KUKA KRL program: e_fraes1.src, e_fraes1.dat

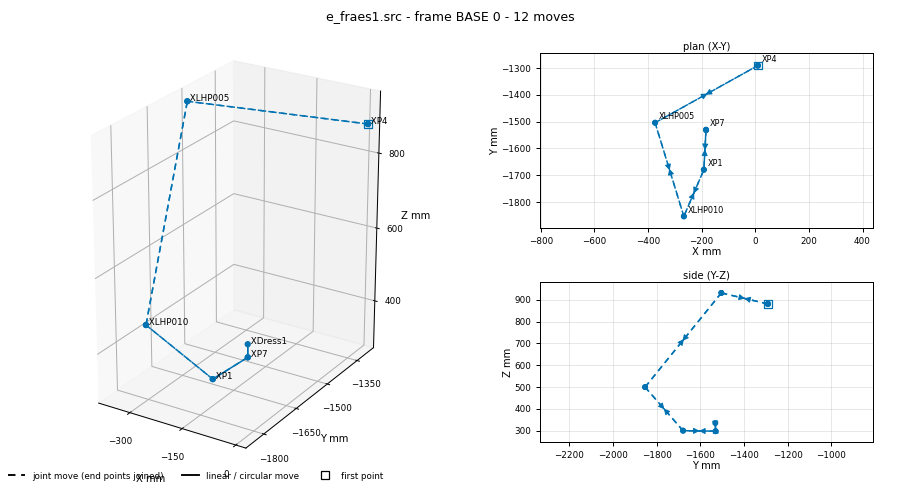
[picture p0: tool path of e_fraes1.src in frame BASE 0, 12 of 12 moves have a stored position in this frame; points joined in program order, loops and branches not executed]
--- e_fraes1.src ---
&ACCESS RVP3
&REL 71
&COMMENT Fresa C1
&PARAM DISKPATH = KRC:\R1\Program
&PARAM TEMPLATE = C:\KRC\Roboter\Template\vorgabe
&PARAM EDITMASK = *
DEF e_fraes1( )
;FOLD INI
   ;FOLD BASISTECH INI
      GLOBAL INTERRUPT DECL 3 WHEN $STOPMESS==TRUE DO IR_STOPM ( )
      INTERRUPT ON 3
      BAS (#INITMOV,0 )
   ;ENDFOLD (BASISTECH INI)
   ;FOLD SPOTTECH INI
      USERSPOT(#INIT)
   ;ENDFOLD (SPOTTECH INI)
   ;FOLD GRIPPERTECH INI
      USER_GRP(0,DUMMY,DUMMY,GDEFAULT)
   ;ENDFOLD (GRIPPERTECH INI)
   ;FOLD USER INI
      ;Make your modifications here

   ;ENDFOLD (USER INI)
;ENDFOLD (INI)

; Estacao P13.060 - Robo R2
; Programa: Fresa C1
; Caracterização dos meios de produção:
; 02/09/2014 09:15 Changes by KUKA Roboter do Brasil

chk_w1_wechs_ok () ;check c1

;FOLD Kollision.Ueberwachung_4_Ein ;%{PE}%MKUKATPUSER
COLLSTOP( 4, 1 ) ;INTERRUPTUEBERWACHT
;ENDFOLD

;FOLD PTP P4 Vel=80 % PDAT6 Tool[1]:GUN C1 Base[0];%{PE}%R 8.2.20,%MKUKATPBASIS,%CMOVE,%VPTP,%P 1:PTP, 2:P4, 3:, 5:80, 7:PDAT6
$BWDSTART=FALSE
PDAT_ACT=PPDAT6
FDAT_ACT=FP4
BAS(#PTP_PARAMS,80)
PTP XP4
;ENDFOLD
;FOLD PTP LHP005 CONT Vel=60 % PDAT2 Tool[1]:GUN C1 Base[0];%{PE}%R 8.2.20,%MKUKATPBASIS,%CMOVE,%VPTP,%P 1:PTP, 2:LHP005, 3:C_DIS, 5:60, 7:PDAT2
$BWDSTART=FALSE
PDAT_ACT=PPDAT2
FDAT_ACT=FLHP005
BAS(#PTP_PARAMS,60)
PTP XLHP005 C_DIS
;ENDFOLD
;FOLD PTP LHP010 CONT Vel= 60 % PDAT3 Tool[1]:GUN C1 Base[0];%{PE}%R 4.1.16,%MKUKATPBASIS,%CMOVE,%VPTP,%P 1:PTP, 2:LHP010, 3:C_PTP, 5:60, 7:PDAT3
$BWDSTART = FALSE
PDAT_ACT=PPDAT3
BAS(#PTP_DAT)
FDAT_ACT=FLHP010
BAS(#FRAMES)
BAS(#VEL_PTP,60)
PTP XLHP010 C_PTP
;ENDFOLD
;FOLD PTP P1 CONT Vel=60 % PDAT1 Tool[1]:GUN C1 Base[0];%{PE}%R 8.2.20,%MKUKATPBASIS,%CMOVE,%VPTP,%P 1:PTP, 2:P1, 3:C_DIS, 5:60, 7:PDAT1
$BWDSTART=FALSE
PDAT_ACT=PPDAT1
FDAT_ACT=FP1
BAS(#PTP_PARAMS,60)
PTP XP1 C_DIS
;ENDFOLD
;FOLD LIN P7 Vel=0.3 m/s CPDAT1 Tool[1]:GUN C1 Base[0];%{PE}%R 8.2.20,%MKUKATPBASIS,%CMOVE,%VLIN,%P 1:LIN, 2:P7, 3:, 5:0.3, 7:CPDAT1
$BWDSTART=FALSE
LDAT_ACT=LCPDAT1
FDAT_ACT=FP7
BAS(#CP_PARAMS,0.3)
LIN XP7
;ENDFOLD

;FOLD ; PONTO DE FRESAGEM;%{PE}%R 4.1.16,%MKUKATPBASIS,%CCOMMENT,%VNORMAL,%P 2:PONTO DE FRESAGEM
;ENDFOLD
;FOLD TIP.LIN_ Dress1, Spot Gun 1 , RETR open , Tool[1], Base[0], EXT.TCP=FALSE;%{PE}%MKUKATPUSER
FDAT_ACT=FDress1
BAS(#FRAMES)
LIN  XDress1
S_ACT.GUN=1
S_ACT.RETR=#opn
S_READY=FALSE
USERSPOT (#DRESS,S_ACT )
WAIT FOR  S_READY
;ENDFOLD

;FOLD LIN LHP020 Vel=0.3 m/s CPDAT16 Tool[1]:GUN C1 Base[0];%{PE}%R 8.2.20,%MKUKATPBASIS,%CMOVE,%VLIN,%P 1:LIN, 2:LHP020, 3:, 5:0.3, 7:CPDAT16
$BWDSTART=FALSE
LDAT_ACT=LCPDAT16
FDAT_ACT=FLHP020
BAS(#CP_PARAMS,0.3)
LIN XLHP020
;ENDFOLD
;FOLD PTP LHP025 CONT Vel= 60 % PDAT7 Tool[1]:GUN C1 Base[0];%{PE}%R 4.1.16,%MKUKATPBASIS,%CMOVE,%VPTP,%P 1:PTP, 2:LHP025, 3:C_PTP, 5:60, 7:PDAT7
$BWDSTART = FALSE
PDAT_ACT=PPDAT7
BAS(#PTP_DAT)
FDAT_ACT=FLHP025
BAS(#FRAMES)
BAS(#VEL_PTP,60)
PTP XLHP025 C_PTP
;ENDFOLD
;FOLD PTP P2 CONT Vel=60 % PDAT4 Tool[1]:GUN C1 Base[0];%{PE}%R 8.2.20,%MKUKATPBASIS,%CMOVE,%VPTP,%P 1:PTP, 2:P2, 3:C_DIS, 5:60, 7:PDAT4
$BWDSTART=FALSE
PDAT_ACT=PPDAT4
FDAT_ACT=FP2
BAS(#PTP_PARAMS,60)
PTP XP2 C_DIS
;ENDFOLD
;FOLD PTP P3 CONT Vel=60 % PDAT5 Tool[1]:GUN C1 Base[0];%{PE}%R 8.2.20,%MKUKATPBASIS,%CMOVE,%VPTP,%P 1:PTP, 2:P3, 3:C_DIS, 5:60, 7:PDAT5
$BWDSTART=FALSE
PDAT_ACT=PPDAT5
FDAT_ACT=FP3
BAS(#PTP_PARAMS,60)
PTP XP3 C_DIS
;ENDFOLD
;FOLD PTP P6 CONT Vel=60 % PDAT9 Tool[1]:GUN C1 Base[0];%{PE}%R 8.2.20,%MKUKATPBASIS,%CMOVE,%VPTP,%P 1:PTP, 2:P6, 3:C_DIS, 5:60, 7:PDAT9
$BWDSTART=FALSE
PDAT_ACT=PPDAT9
FDAT_ACT=FP6
BAS(#PTP_PARAMS,60)
PTP XP6 C_DIS
;ENDFOLD
;FOLD PTP pTEST_WELD PDAT10 SPOT Gun= 1 RETR OPN PgNo1= 251 ACTIVE= 1 Tool[1]:GUN C1 Base[0];%{PE}%R 4.1.12,%MKUKATPSPOT,%CSPOT,%VPTP,%P 1:PTP, 2:pTEST_WELD, 3:, 5:60, 7:PDAT10, 10:1, 12:#FIRST, 14:#OPN, 16:251, 18:1, 20:0, 22:0, 24:1, 25:NORMAL
$BWDSTART = FALSE
PDAT_ACT=PPDAT10
BAS(#PTP_DAT)
FDAT_ACT=FpTEST_WELD
BAS(#FRAMES)
BAS(#VEL_PTP,PPDAT10.VEL)
S_ACT.GUN=1
S_ACT.PAIR=SDEFAULT.PAIR
S_ACT.RETR=#OPN
S_ACT.CLO_TM=1
S_ACT.PGNO1=251
S_ACT.PGNO2=SDEFAULT.PGNO2
S_ACT.PRESS1=SDEFAULT.PRESS1
S_ACT.PRESS2=SDEFAULT.PRESS2
S_READY=FALSE
PTP XpTEST_WELD
USERSPOT(#SPOT, S_ACT)
WAIT FOR S_READY
;ENDFOLD

;FOLD Kollision.Ueberwachung_4_Aus ;%{PE}%MKUKATPUSER
COLLSTOP( 4, 2 )
;ENDFOLD

END

--- e_fraes1.dat ---
&ACCESS RVP3
&REL 71
&COMMENT Fresa C1
&PARAM DISKPATH = KRC:\R1\Program
&PARAM TEMPLATE = C:\KRC\Roboter\Template\vorgabe
&PARAM EDITMASK = *
DEFDAT  e_fraes1
;FOLD EXTERNAL DECLARATIONS;%{PE}%MKUKATPBASIS,%CEXT,%VCOMMON,%P
;FOLD GRIPPERTECH EXT
EXT  H50 (INT  :IN,INT  :IN,INT  :IN,GRP_TYP  :IN )
;ENDFOLD (GRIPPERTECH EXT)
;FOLD SPOTTECH EXT
EXT  USERSPOT (S_COMMAND  :IN,SPOT_TYPE  :IN )
;ENDFOLD (SPOTTECH EXT)
;FOLD BASISTECH EXT;%{PE}%MKUKATPBASIS,%CEXT,%VEXT,%P
EXT  BAS (BAS_COMMAND  :IN,REAL  :IN )
DECL INT SUCCESS
;ENDFOLD (BASISTECH EXT)
;FOLD USER EXT;%{E}%MKUKATPUSER,%CEXT,%VEXT,%P
;Make your modifications here

;ENDFOLD (USER EXT)
;ENDFOLD (EXTERNAL DECLARATIONS)

DECL E6POS XLHP010={X -266.548096,Y -1853.20605,Z 499.976013,A 107.124496,B 39.7114487,C 7.39129782,S 18,T 42,E1 0.0,E2 0.0,E3 0.0,E4 0.0,E5 0.0,E6 0.0}
DECL FDAT FLHP010={TOOL_NO 1,BASE_NO 0,IPO_FRAME #BASE}
DECL PDAT PPDAT2={VEL 80.0,ACC 100.0,APO_DIST 20.0,APO_MODE #CDIS}
DECL PDAT PPDAT3={VEL 100.0,ACC 100.0,APO_DIST 10.0}
DECL FDAT FDress1={TOOL_NO 1,BASE_NO 0,IPO_FRAME #BASE}
DECL E6POS XDress1={X -183.147598,Y -1531.61096,Z 335.393188,A 96.1598816,B 0.990136683,C 0.264630109,S 18,T 34,E1 0.0,E2 0.0,E3 0.0,E4 0.0,E5 0.0,E6 0.0}
DECL E6POS XLHP025={X -191.917496,Y -1679.34094,Z 300.446106,A 96.1167603,B 18.2161503,C 4.02709389,S 18,T 34,E1 0.0,E2 0.0,E3 0.0,E4 0.0,E5 0.0,E6 0.0}
DECL FDAT FLHP025={TOOL_NO 1,BASE_NO 0,IPO_FRAME #BASE}
DECL PDAT PPDAT7={VEL 100.0,ACC 100.0,APO_DIST 10.0}
DECL E6POS XLHP020={X -183.854095,Y -1530.21204,Z 298.03421,A 94.9578705,B -2.47679901,C -0.118712999,S 18,T 34,E1 0.0,E2 0.0,E3 0.0,E4 0.0,E5 0.0,E6 0.0}
DECL FDAT FLHP020={TOOL_NO 1,BASE_NO 0,IPO_FRAME #BASE}
DECL LDAT LCPDAT16={VEL 2.0,ACC 100.0,APO_DIST 5.0,APO_FAC 50.0}
DECL E6POS XPTEST_WELD={X 9.70383453,Y -1290.66699,Z 880.833679,A -89.7398682,B -10.2741604,C 0.05478286,S 18,T 2,E1 0.0,E2 0.0,E3 0.0,E4 0.0,E5 0.0,E6 0.0}
DECL FDAT FpTEST_WELD={TOOL_NO 1,BASE_NO 0,IPO_FRAME #BASE}
DECL PDAT PPDAT10={VEL 100.0,ACC 100.0,APO_DIST 100.0}
DECL E6POS XLHP005={X -373.799011,Y -1504.00696,Z 931.286621,A 174.520996,B 1.51326394,C 20.2021408,S 18,T 42,E1 0.0,E2 0.0,E3 0.0,E4 0.0,E5 0.0,E6 0.0}
DECL FDAT FLHP005={TOOL_NO 1,BASE_NO 0,IPO_FRAME #BASE}
DECL BASIS_SUGG_T LAST_BASIS={POINT1[] "P7                      ",POINT2[] "P7                      ",CP_PARAMS[] "CPDAT1                  ",PTP_PARAMS[] "PDAT9                   ",CONT[] "                        ",CP_VEL[] "0.3                     ",PTP_VEL[] "60                      ",SYNC_PARAMS[] "SYNCDAT                 ",SPL_NAME[] "S0                      "}
DECL E6POS XP1={X -191.919296,Y -1679.37305,Z 300.448792,A 96.1213074,B 18.2176094,C 4.0277338,S 18,T 34,E1 0.0,E2 0.0,E3 0.0,E4 0.0,E5 0.0,E6 0.0}
DECL FDAT FP1={TOOL_NO 1,BASE_NO 0,IPO_FRAME #BASE,POINT2[] " ",TQ_STATE FALSE}
DECL PDAT PPDAT1={VEL 100.0,ACC 100.0,APO_DIST 10.0,APO_MODE #CDIS,GEAR_JERK 50.0}
DECL E6POS XP2={X -266.550995,Y -1853.18994,Z 499.962189,A 107.124199,B 39.7108192,C 7.39097309,S 18,T 42,E1 0.0,E2 0.0,E3 0.0,E4 0.0,E5 0.0,E6 0.0}
DECL FDAT FP2={TOOL_NO 1,BASE_NO 0,IPO_FRAME #BASE,POINT2[] " ",TQ_STATE FALSE}
DECL PDAT PPDAT4={VEL 100.0,ACC 100.0,APO_DIST 10.0,APO_MODE #CDIS,GEAR_JERK 50.0}
DECL E6POS XP3={X -373.798004,Y -1503.99805,Z 931.282593,A 174.520905,B 1.51325798,C 20.2017708,S 18,T 42,E1 0.0,E2 0.0,E3 0.0,E4 0.0,E5 0.0,E6 0.0}
DECL FDAT FP3={TOOL_NO 1,BASE_NO 0,IPO_FRAME #BASE,POINT2[] " ",TQ_STATE FALSE}
DECL PDAT PPDAT5={VEL 100.0,ACC 100.0,APO_DIST 10.0,APO_MODE #CDIS,GEAR_JERK 50.0}
DECL E6POS XP4={X 9.70852661,Y -1290.67603,Z 880.838196,A -89.7397919,B -10.2745199,C 0.0549346097,S 18,T 10,E1 0.0,E2 0.0,E3 0.0,E4 0.0,E5 0.0,E6 0.0}
DECL FDAT FP4={TOOL_NO 1,BASE_NO 0,IPO_FRAME #BASE,POINT2[] " ",TQ_STATE FALSE}
DECL PDAT PPDAT6={VEL 100.0,ACC 100.0,APO_DIST 10.0,APO_MODE #CDIS,GEAR_JERK 50.0}
DECL E6POS XP6={X 9.69707203,Y -1290.64697,Z 880.824219,A -89.7402267,B -10.2734003,C 0.0546588488,S 18,T 2,E1 0.0,E2 0.0,E3 0.0,E4 0.0,E5 0.0,E6 0.0}
DECL FDAT FP6={TOOL_NO 1,BASE_NO 0,IPO_FRAME #BASE,POINT2[] " ",TQ_STATE FALSE}
DECL PDAT PPDAT9={VEL 100.0,ACC 100.0,APO_DIST 20.0,APO_MODE #CDIS,GEAR_JERK 50.0}
DECL E6POS XP7={X -183.848907,Y -1530.14197,Z 298.066315,A 94.9547272,B -1.64593899,C -0.0469314381,S 18,T 34,E1 0.0,E2 0.0,E3 0.0,E4 0.0,E5 0.0,E6 0.0}
DECL FDAT FP7={TOOL_NO 1,BASE_NO 0,IPO_FRAME #BASE,POINT2[] " ",TQ_STATE FALSE}
DECL LDAT LCPDAT1={VEL 2.0,ACC 100.0,APO_DIST 100.0,APO_FAC 50.0,AXIS_VEL 100.0,AXIS_ACC 100.0,ORI_TYP #VAR,CIRC_TYP #BASE,JERK_FAC 50.0,GEAR_JERK 50.0,EXAX_IGN 0}
ENDDAT
